(*
SPDX-FileCopyrightText: © 2026 Oleksandr Tiutyk <trofimich@gmail.com>
SPDX-License-Identifier: MIT
License: https://opensource.org/license/mit
*)

INTERFACE IActionPermissionProvider EXTENDS IObject

METHOD RequestActionPermission : BOOL
VAR_INPUT
	actionDescriptor : INamed;
	requestingObject : IObject;
END_VAR
VAR_IN_OUT
	rejectReason : WSTRING(255);
END_VAR
END_METHOD

END_INTERFACE

(* stored: Version 1.1.0.1
   Itf IActionPermissionProvider: Id {11122ffc-a610-4022-99ee-4c4322cf06fe}
   Method RequestActionPermission: Id {f812615f-fe7b-472c-83d6-4941a1e729d2} *)
